TYPE DUT_LogowanieBledow_ZdarzenieOpis :
STRUCT
	iIdZdarzenia							: INT;
	sOpis									: STRING;
END_STRUCT
END_TYPE

(* stored: Version 1.1.0.1, ProductVersion 3.1.4024.11
   DUT DUT_LogowanieBledow_ZdarzenieOpis: Id {f7ba6a38-77f4-403f-a44d-e9677655cd1b} *)
